TYPE ST_AlpacaPutNoArgs EXTENDS ST_AlpacaPutRequest:
STRUCT
    // just for the sake of semantics, our 'No args' structure extends
    // our common "put" request structure, but it doesn't add any members.
END_STRUCT
END_TYPE

(* stored: Version 1.1.0.1, ProductVersion 3.1.4024.12
   DUT ST_AlpacaPutNoArgs: Id {a447eb8f-0556-423f-93df-a73db172c007} *)
